// TIA Portal V20 export
DATA_BLOCK "PM6"   // DB280
// stored: MemoryReserve 100
   VAR
      "SIDE TAPE FIX STAGE CLOSE" : Bool;
      "SIDE TAPE FIX STAGE OPEN" : Bool;
      "SIDE TAPE Attachment LEFT FORWARD" : Bool;
      "SIDE TAPE Attachment LEFT BACKWARD" : Bool;
      "SIDE TAPE Attachment RIGHT FORWARD" : Bool;
      "SIDE TAPE Attachment RIGHT BACKWARD" : Bool;
      "SIDE TAPE Attachment BTM FORWARD" : Bool;
      "SIDE TAPE Attachment BTM BACKWARD" : Bool;
      SPARE : Bool;
      SPARE_1 : Bool;
      SPARE_2 : Bool;
      SPARE_3 : Bool;
      SPARE_4 : Bool;
      SPARE_5 : Bool;
      SPARE_6 : Bool;
      SPARE_7 : Bool;
   END_VAR
BEGIN
END_DATA_BLOCK
